FUNCTION_BLOCK XCBR_Logic (* Basic Function Block Type *)
  (* Standard: 61499-2 *)
  (* Version 0.0, 12/11/2023, Cheyan, Schneider Electric, Template *)
  PACKAGE Main;
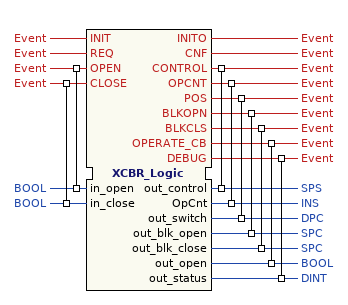
  EVENT_INPUT
    INIT; (* Initialization Request *)
    REQ; (* Normal Execution Request *)
    OPEN WITH in_open;
    CLOSE WITH in_close;
  END_EVENT
  EVENT_OUTPUT
    INITO; (* Initialization Confirm *)
    CNF; (* Execution Confirmation *)
    CONTROL WITH out_control;
    OPCNT WITH OpCnt;
    POS WITH out_switch;
    BLKOPN WITH out_blk_open;
    BLKCLS WITH out_blk_close;
    OPERATE_CB WITH out_open;
    DEBUG WITH out_status;
  END_EVENT
  VAR_INPUT
    in_open : BOOL; (* Input event qualifier *)
    in_close : BOOL;
  END_VAR
  VAR_OUTPUT
    out_control : SPS;
    OpCnt : INS;
    out_switch : DPC;
    out_blk_open : SPC;
    out_blk_close : SPC;
    out_open : BOOL;
    out_status : DINT;
  END_VAR
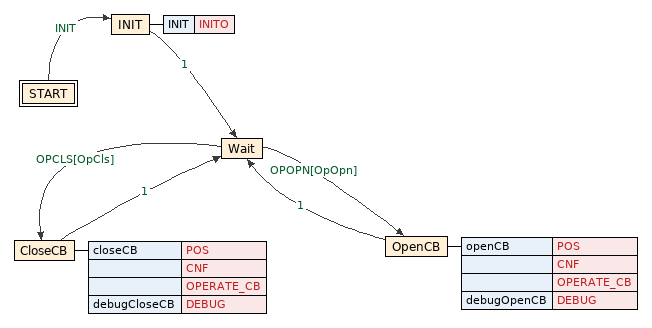
  EC_STATES
    START; (* Initial State *)
    INIT : INIT -> INITO; (* Initialization *)
    Wait; (* Normal execution *)
    OpenCB : openCB -> POS, -> CNF, -> OPERATE_CB, debugOpenCB -> DEBUG;
    CloseCB : closeCB -> POS, -> CNF, -> OPERATE_CB, debugCloseCB -> DEBUG;
  END_STATES
  EC_TRANSITIONS
    START TO INIT := INIT;
    INIT TO Wait := 1;
    Wait TO OpenCB := OPOPN[OpOpn];
    OpenCB TO Wait := 1;
    Wait TO CloseCB := OPCLS[OpCls];
    CloseCB TO Wait := 1;
  END_TRANSITIONS
  ALGORITHM INIT IN ST: (* Initialization algorithm Setting the initial position of the CB to the "Closed" state stVal is a coded Enum: "1:intermediate-state 2:off 3:on 4:bad-state" *)
;

out_switch.stVal := Main.stVal#item3;
  END_ALGORITHM
  ALGORITHM REQ IN ST: (* Normally executed algorithm *)
;
  END_ALGORITHM
  ALGORITHM openCB IN ST: (* To open the CB, set Pos_stVal to false Setting the initial position of the CB to the "opened" state stVal is a coded Enum: "1:intermediate-state 2:off 3:on 4:bad-state" *)
;

out_switch.stVal := Main.stVal#item2;

// Open the CB in our plant model
out_open := TRUE;
  END_ALGORITHM
  ALGORITHM closeCB IN ST: (* To close the CB, set Pos_stVal to true Setting the initial position of the CB to the "Closed" state stVal is a coded Enum: "1:intermediate-state 2:off 3:on 4:bad-state" *)
;

out_switch.stVal := Main.stVal#item3;

// Close the CB in our plant model
out_open := FALSE;
  END_ALGORITHM
  ALGORITHM debugOpenCB IN ST:
;

debug_Pos_stVal := 2;
  END_ALGORITHM
  ALGORITHM debugCloseCB IN ST:
;

debug_Pos_stVal := 3;
  END_ALGORITHM
END_FUNCTION_BLOCK
